ABB RobotStudio station: harithagracy_final.rsstn

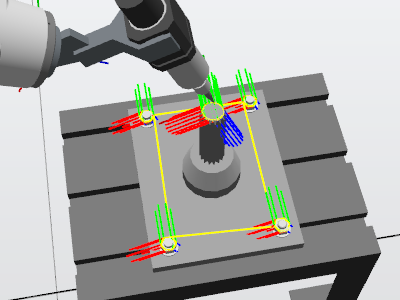
Station harithagracy_final (saved by RobotStudio 22.3.10141.1)
Controller Controller11
  mechanical unit ROB_1: IRB1520ID_4_150__02, 6 joints, base frame (0, 0, 0) mm
Layout (positions relative to the parent item):
  - IRB1520ID_4_150__02 [mechanism, from Robots\IRB1520ID_4_150_G_02.rslib] at (0, 0, 0) mm; joint values [0.0152, 0.1229, 0.5695, 0.0782, -0.1693, -0.0695] (rad or m)
  - MyTool [mechanism, from Training Objects\myTool.rslib] at (1089.61, 13.93, 630.91) mm, rotated rx 180 ry 60 rz 180 deg
  - table_and_fixture_140 [part, from Training Objects\propeller_table.rslib] at (1043.36, -175, 17.55) mm
Attachment: MyTool is attached to IRB1520ID_4_150__02 / Link6
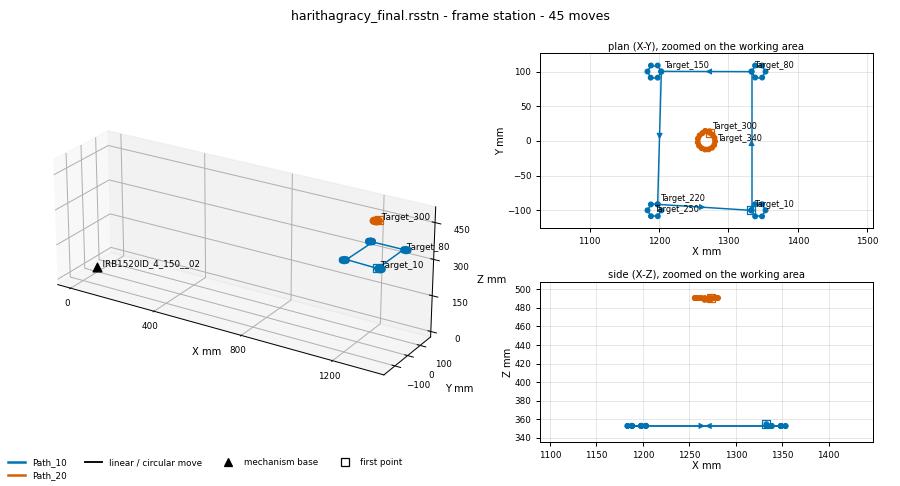
[picture p0: tool path of harithagracy_final.rsstn in frame station, 45 of 45 moves have a stored position in this frame; points joined in program order, loops and branches not executed]
Targets, tools, work objects and paths stored in the station, written as RAPID:
! task T_ROB1
MODULE CalibData
  PERS tooldata MyTool:=[TRUE,[[31.792631019,0,229.638935148],[0.945518576,0,0.325568154,0]],[1,[0,0,1],[1,0,0,0],0,0,0]];
ENDMODULE

! task T_ROB1
MODULE Module1
  CONST robtarget Target_10:=[[1332.924046806,-99.901116574,354.773786223],[0.190807747,-0.000000001,0.981627426,0.000000001],[-1,-1,0,1],[9E+09,9E+09,9E+09,9E+09,9E+09,9E+09]];
  CONST robtarget Target_20:=[[1338.536067515,-108.623502158,352.735405433],[0.190806659,0.000000047,0.981627638,0.000000014],[-1,-1,0,1],[9E+09,9E+09,9E+09,9E+09,9E+09,9E+09]];
  CONST robtarget Target_30:=[[1348.455004827,-108.623495689,352.735420125],[0.190806668,0.00000004,0.981627636,0.000000009],[-1,-1,0,1],[9E+09,9E+09,9E+09,9E+09,9E+09,9E+09]];
  CONST robtarget Target_40:=[[1353.51710265,-99.906819828,352.735392671],[0.190806553,0.000000024,0.981627658,0],[-1,-1,0,1],[9E+09,9E+09,9E+09,9E+09,9E+09,9E+09]];
  CONST robtarget Target_50:=[[1348.531058556,-91.168690385,352.90628556],[0.19080656,0.000000021,0.981627657,-0.000000007],[-1,-1,0,1],[9E+09,9E+09,9E+09,9E+09,9E+09,9E+09]];
  CONST robtarget Target_60:=[[1338.353068386,-91.16869192,352.906259589],[0.190806544,0.000000028,0.98162766,-0.000000002],[-1,-1,0,1],[9E+09,9E+09,9E+09,9E+09,9E+09,9E+09]];
  CONST robtarget Target_70:=[[1333.369050893,-99.863781416,352.90625685],[0.190806109,0.00000003,0.981627744,-0.000000004],[-1,-1,0,1],[9E+09,9E+09,9E+09,9E+09,9E+09,9E+09]];
  CONST robtarget Target_80:=[[1333.369054607,100.0996057,352.906282296],[0.190805935,0.00000002,0.981627778,-0.000000009],[0,0,-1,1],[9E+09,9E+09,9E+09,9E+09,9E+09,9E+09]];
  CONST robtarget Target_90:=[[1338.549046447,91.330040115,352.906243486],[0.190805129,0.000000015,0.981627935,-0.000000006],[0,0,-1,1],[9E+09,9E+09,9E+09,9E+09,9E+09,9E+09]];
  CONST robtarget Target_100:=[[1348.629984002,91.330033876,352.906247133],[0.190805045,0.000000017,0.981627951,-0.000000005],[0,0,-1,1],[9E+09,9E+09,9E+09,9E+09,9E+09,9E+09]];
  CONST robtarget Target_110:=[[1353.489085679,99.906654409,352.906268106],[0.190804956,0.000000021,0.981627969,0],[0,0,-1,1],[9E+09,9E+09,9E+09,9E+09,9E+09,9E+09]];
  CONST robtarget Target_120:=[[1348.546066846,108.622506471,352.885511001],[0.190804528,0.000000005,0.981628052,0],[0,0,-1,1],[9E+09,9E+09,9E+09,9E+09,9E+09,9E+09]];
  CONST robtarget Target_130:=[[1338.417093775,108.622495135,352.885505396],[0.190804431,0.000000008,0.981628071,0],[0,0,-1,1],[9E+09,9E+09,9E+09,9E+09,9E+09,9E+09]];
  CONST robtarget Target_140:=[[1333.37205346,99.788553235,352.885529006],[0.190804152,0.000000009,0.981628125,0.000000006],[0,0,-1,1],[9E+09,9E+09,9E+09,9E+09,9E+09,9E+09]];
  CONST robtarget Target_150:=[[1203.12409131,100.220808495,352.885516231],[0.190803949,0.000000011,0.981628164,0.000000004],[0,0,-1,1],[9E+09,9E+09,9E+09,9E+09,9E+09,9E+09]];
  CONST robtarget Target_160:=[[1198.185025055,108.617502854,352.885533365],[0.190803859,0.000000023,0.981628182,0.000000014],[0,0,-1,1],[9E+09,9E+09,9E+09,9E+09,9E+09,9E+09]];
  CONST robtarget Target_170:=[[1188.446086111,108.61750794,352.885518095],[0.19080385,0.00000002,0.981628184,0.000000014],[0,0,-1,1],[9E+09,9E+09,9E+09,9E+09,9E+09,9E+09]];
  CONST robtarget Target_180:=[[1183.411995563,100.014506274,352.885514495],[0.190803746,0.000000018,0.981628204,0.000000014],[0,0,-1,1],[9E+09,9E+09,9E+09,9E+09,9E+09,9E+09]];
  CONST robtarget Target_190:=[[1188.06105093,91.14996766,353.102010282],[0.190802255,0.000000008,0.981628494,0.00000002],[0,0,-1,1],[9E+09,9E+09,9E+09,9E+09,9E+09,9E+09]];
  CONST robtarget Target_200:=[[1198.115984646,91.14997454,353.102001135],[0.190802253,0.000000013,0.981628494,0.000000025],[0,0,-1,1],[9E+09,9E+09,9E+09,9E+09,9E+09,9E+09]];
  CONST robtarget Target_210:=[[1203.421049436,99.621912059,353.102013314],[0.190801872,-0.000000005,0.981628568,0.000000013],[0,0,-1,1],[9E+09,9E+09,9E+09,9E+09,9E+09,9E+09]];
  CONST robtarget Target_220:=[[1198.097969428,-91.440610478,352.955677838],[0.190800632,-0.000000022,0.981628809,-0.000000002],[-1,-1,0,1],[9E+09,9E+09,9E+09,9E+09,9E+09,9E+09]];
  CONST robtarget Target_230:=[[1188.385983378,-91.440612767,352.955671893],[0.190800549,-0.000000022,0.981628825,-0.000000001],[-1,-1,0,1],[9E+09,9E+09,9E+09,9E+09,9E+09,9E+09]];
  CONST robtarget Target_240:=[[1183.475073313,-99.92918803,352.955726223],[0.190800374,-0.000000034,0.981628859,-0.000000009],[-1,-1,0,1],[9E+09,9E+09,9E+09,9E+09,9E+09,9E+09]];
  CONST robtarget Target_250:=[[1188.462071492,-108.375988296,352.955716254],[0.190800062,-0.000000043,0.98162892,-0.000000004],[-1,-1,0,1],[9E+09,9E+09,9E+09,9E+09,9E+09,9E+09]];
  CONST robtarget Target_260:=[[1198.351060599,-108.375991624,352.955682567],[0.190800042,-0.000000041,0.981628924,0],[-1,-1,0,1],[9E+09,9E+09,9E+09,9E+09,9E+09,9E+09]];
  CONST robtarget Target_270:=[[1203.36607102,-100.060801151,352.955685774],[0.190799918,-0.000000029,0.981628948,0.000000007],[-1,-1,0,1],[9E+09,9E+09,9E+09,9E+09,9E+09,9E+09]];
  CONST robtarget Target_280:=[[1198.251066287,-91.352908584,352.955719652],[0.190799466,-0.00000001,0.981629036,0.000000012],[-1,-1,0,1],[9E+09,9E+09,9E+09,9E+09,9E+09,9E+09]];
  CONST robtarget Target_290:=[[1333.058061673,-100.004400902,352.955724265],[0.190798868,-0.000000005,0.981629152,0.00000001],[-1,-1,0,1],[9E+09,9E+09,9E+09,9E+09,9E+09,9E+09]];
  CONST robtarget Target_300:=[[1272.877007141,11.820189365,490.550894391],[0.190798043,0.000000003,0.981629312,0.000000018],[0,0,-1,1],[9E+09,9E+09,9E+09,9E+09,9E+09,9E+09]];
  CONST robtarget Target_310:=[[1277.295045776,8.963074457,490.550919493],[0.190797854,0.000000002,0.981629349,0.000000018],[0,0,-1,1],[9E+09,9E+09,9E+09,9E+09,9E+09,9E+09]];
  CONST robtarget Target_320:=[[1280.04804639,4.443500887,490.550889318],[0.190797353,0.000000002,0.981629446,0.000000017],[0,0,-1,1],[9E+09,9E+09,9E+09,9E+09,9E+09,9E+09]];
  CONST robtarget Target_330:=[[1280.846049267,-0.69278741,490.550917172],[0.190797368,0.000000002,0.981629443,0.000000017],[-1,-1,0,1],[9E+09,9E+09,9E+09,9E+09,9E+09,9E+09]];
  CONST robtarget Target_340:=[[1279.649052695,-5.722865911,490.550897036],[0.190797358,0.000000002,0.981629445,0.000000018],[-1,-1,0,1],[9E+09,9E+09,9E+09,9E+09,9E+09,9E+09]];
  CONST robtarget Target_350:=[[1276.345038332,-9.817636042,490.550864439],[0.19079722,0.000000001,0.981629472,0.000000018],[-1,-1,0,1],[9E+09,9E+09,9E+09,9E+09,9E+09,9E+09]];
  CONST robtarget Target_360:=[[1271.563092559,-12.084020458,490.550898195],[0.190797134,0.000000002,0.981629489,0.000000019],[-1,-1,0,1],[9E+09,9E+09,9E+09,9E+09,9E+09,9E+09]];
  CONST robtarget Target_370:=[[1266.371043262,-12.340000508,490.550890824],[0.19079682,0.000000006,0.98162955,0.000000022],[-1,-1,0,1],[9E+09,9E+09,9E+09,9E+09,9E+09,9E+09]];
  CONST robtarget Target_380:=[[1261.525064206,-10.462289676,490.550892331],[0.190796734,0.000000006,0.981629567,0.000000022],[-1,-1,0,1],[9E+09,9E+09,9E+09,9E+09,9E+09,9E+09]];
  CONST robtarget Target_390:=[[1257.767002799,-6.91063053,490.550902041],[0.190796538,0.000000005,0.981629605,0.000000022],[-1,-1,0,1],[9E+09,9E+09,9E+09,9E+09,9E+09,9E+09]];
  CONST robtarget Target_400:=[[1255.872050443,-2.002559039,490.550904643],[0.190796442,0.000000005,0.981629624,0.000000022],[-1,-1,0,1],[9E+09,9E+09,9E+09,9E+09,9E+09,9E+09]];
  CONST robtarget Target_410:=[[1256.13802064,3.251771994,490.550927585],[0.190796366,0.000000006,0.981629638,0.000000022],[0,0,-1,1],[9E+09,9E+09,9E+09,9E+09,9E+09,9E+09]];
  CONST robtarget Target_420:=[[1258.518020461,7.943842238,490.55090574],[0.190796355,0.000000007,0.98162964,0.000000023],[0,0,-1,1],[9E+09,9E+09,9E+09,9E+09,9E+09,9E+09]];
  CONST robtarget Target_430:=[[1262.599986723,11.26235147,490.550893658],[0.190796326,0.000000007,0.981629646,0.000000023],[0,0,-1,1],[9E+09,9E+09,9E+09,9E+09,9E+09,9E+09]];
  CONST robtarget Target_440:=[[1266.551051866,14.43843955,488.550888807],[0.190796224,0.000000005,0.981629666,0.000000022],[0,0,-1,1],[9E+09,9E+09,9E+09,9E+09,9E+09,9E+09]];
  CONST robtarget Target_450:=[[1272.581032519,13.927840241,488.550917974],[0.19079614,0.000000003,0.981629682,0.00000002],[0,0,-1,1],[9E+09,9E+09,9E+09,9E+09,9E+09,9E+09]];
  PROC Path_10()
    MoveL Target_10,v1000,fine,MyTool\WObj:=wobj0;
    MoveL Target_20,v1000,fine,MyTool\WObj:=wobj0;
    MoveL Target_30,v1000,fine,MyTool\WObj:=wobj0;
    MoveL Target_40,v1000,fine,MyTool\WObj:=wobj0;
    MoveL Target_50,v1000,fine,MyTool\WObj:=wobj0;
    MoveL Target_60,v1000,fine,MyTool\WObj:=wobj0;
    MoveL Target_70,v1000,fine,MyTool\WObj:=wobj0;
    MoveL Target_80,v1000,fine,MyTool\WObj:=wobj0;
    MoveL Target_90,v1000,fine,MyTool\WObj:=wobj0;
    MoveL Target_100,v1000,fine,MyTool\WObj:=wobj0;
    MoveL Target_110,v1000,fine,MyTool\WObj:=wobj0;
    MoveL Target_120,v1000,fine,MyTool\WObj:=wobj0;
    MoveL Target_130,v1000,fine,MyTool\WObj:=wobj0;
    MoveL Target_140,v1000,fine,MyTool\WObj:=wobj0;
    MoveL Target_150,v1000,fine,MyTool\WObj:=wobj0;
    MoveL Target_160,v1000,fine,MyTool\WObj:=wobj0;
    MoveL Target_170,v1000,fine,MyTool\WObj:=wobj0;
    MoveL Target_180,v1000,fine,MyTool\WObj:=wobj0;
    MoveL Target_190,v1000,fine,MyTool\WObj:=wobj0;
    MoveL Target_200,v1000,fine,MyTool\WObj:=wobj0;
    MoveL Target_210,v1000,fine,MyTool\WObj:=wobj0;
    MoveL Target_220,v1000,fine,MyTool\WObj:=wobj0;
    MoveL Target_230,v1000,fine,MyTool\WObj:=wobj0;
    MoveL Target_240,v1000,fine,MyTool\WObj:=wobj0;
    MoveL Target_250,v1000,fine,MyTool\WObj:=wobj0;
    MoveL Target_260,v1000,fine,MyTool\WObj:=wobj0;
    MoveL Target_270,v1000,fine,MyTool\WObj:=wobj0;
    MoveL Target_280,v1000,fine,MyTool\WObj:=wobj0;
    MoveL Target_290,v1000,fine,MyTool\WObj:=wobj0;
  ENDPROC
  PROC Path_20()
    MoveL Target_300,v1000,z100,MyTool\WObj:=wobj0;
    MoveL Target_310,v1000,z100,MyTool\WObj:=wobj0;
    MoveL Target_320,v1000,z100,MyTool\WObj:=wobj0;
    MoveL Target_330,v1000,z100,MyTool\WObj:=wobj0;
    MoveL Target_340,v1000,z100,MyTool\WObj:=wobj0;
    MoveL Target_350,v1000,z100,MyTool\WObj:=wobj0;
    MoveL Target_360,v1000,z100,MyTool\WObj:=wobj0;
    MoveL Target_370,v1000,z100,MyTool\WObj:=wobj0;
    MoveL Target_380,v1000,z100,MyTool\WObj:=wobj0;
    MoveL Target_390,v1000,z100,MyTool\WObj:=wobj0;
    MoveL Target_400,v1000,z100,MyTool\WObj:=wobj0;
    MoveL Target_410,v1000,z100,MyTool\WObj:=wobj0;
    MoveL Target_420,v1000,z100,MyTool\WObj:=wobj0;
    MoveL Target_430,v1000,z100,MyTool\WObj:=wobj0;
    MoveL Target_440,v1000,z100,MyTool\WObj:=wobj0;
    MoveL Target_450,v1000,z100,MyTool\WObj:=wobj0;
  ENDPROC
  PROC Path_30()
    Path_10;
    Path_20;
  ENDPROC
ENDMODULE

